// TIA Portal V18 export
FUNCTION "ERRORS_WARNINGS_main" : Void   // FC32, FBD
{ S7_Optimized_Access := 'TRUE' }
VERSION : 0.1
// stored: AutoNumber true, IsIECCheckEnabled false, SetENOAutomatically false, UDAEnableTagReadback false
   VAR_TEMP
      er_count : Int;
      wn_count : Int;
      loc_count : Int;
      loc_c : Bool;
   END_VAR
BEGIN

REGION Network 1
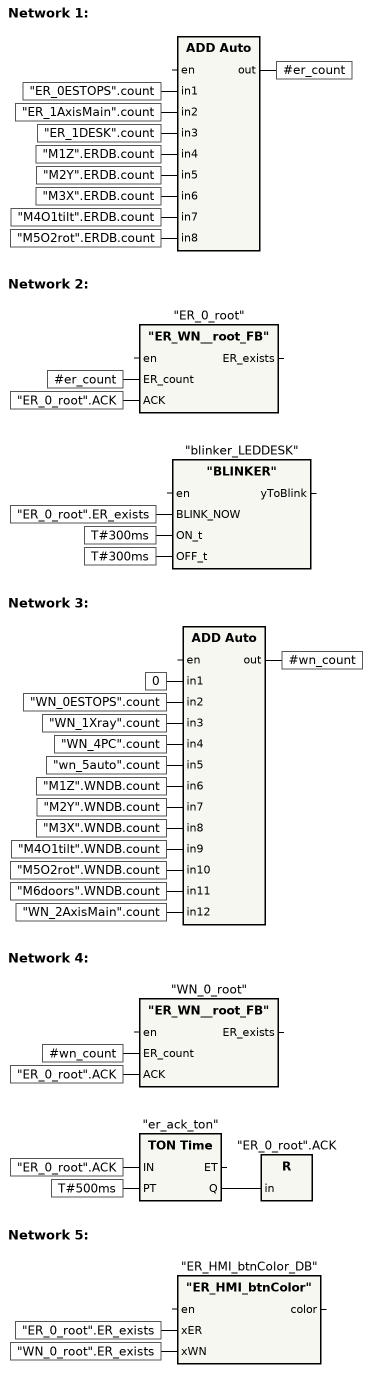
   #er_count := "ER_0ESTOPS".count + "ER_1AxisMain".count + "ER_1DESK".count + "M1Z".ERDB.count + "M2Y".ERDB.count + "M3X".ERDB.count + "M4O1tilt".ERDB.count + "M5O2rot".ERDB.count;
END_REGION

REGION Network 2
   "ER_0_root"(ER_count := #er_count, ACK := "ER_0_root".ACK);   // "ER_WN__root_FB"
   "blinker_LEDDESK"(BLINK_NOW := "ER_0_root".ER_exists, ON_t := T#300ms, OFF_t := T#300ms);   // "BLINKER"
END_REGION

REGION Network 3
   #wn_count := 0 + "WN_0ESTOPS".count + "WN_1Xray".count + "WN_4PC".count + "wn_5auto".count + "M1Z".WNDB.count + "M2Y".WNDB.count + "M3X".WNDB.count + "M4O1tilt".WNDB.count + "M5O2rot".WNDB.count + "M6doors".WNDB.count + "WN_2AxisMain".count;
END_REGION

REGION Network 4
   "WN_0_root"(ER_count := #wn_count, ACK := "ER_0_root".ACK);   // "ER_WN__root_FB"
   "er_ack_ton".TON(IN := "ER_0_root".ACK, PT := T#500ms);
   IF "er_ack_ton".Q THEN "ER_0_root".ACK := FALSE; END_IF;
END_REGION

REGION Network 5
   "ER_HMI_btnColor_DB"(xER := "ER_0_root".ER_exists, xWN := "WN_0_root".ER_exists);   // "ER_HMI_btnColor"
END_REGION

REGION Network 6
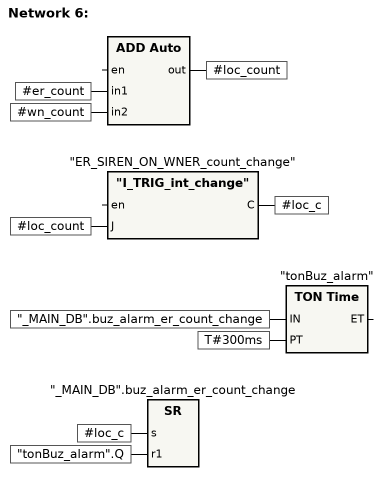
   #loc_count := #er_count + #wn_count;
   "ER_SIREN_ON_WNER_count_change"(J := #loc_count, C => #loc_c);   // "I_TRIG_int_change"
   "tonBuz_alarm".TON(IN := "_MAIN_DB".buz_alarm_er_count_change, PT := T#300ms);
   IF #loc_c THEN
       "_MAIN_DB".buz_alarm_er_count_change := TRUE;   // SR flip-flop
   END_IF;
   IF "tonBuz_alarm".Q THEN "_MAIN_DB".buz_alarm_er_count_change := FALSE; END_IF;
END_REGION
END_FUNCTION
